{attribute 'qualified_only'}
{attribute 'strict'}
{attribute 'to_string'}
TYPE E_RecipeRunETMode :
(
	None := 0,
	Ramp := 1,
	Hold := 2
);
END_TYPE

(* stored: Version 1.1.0.1, ProductVersion 3.1.4026.11
   DUT E_RecipeRunETMode: Id {88628f77-d0bd-459d-a557-53750e6e0c09} *)
